Universal Robots PolyScope program: venosa draft3.urp

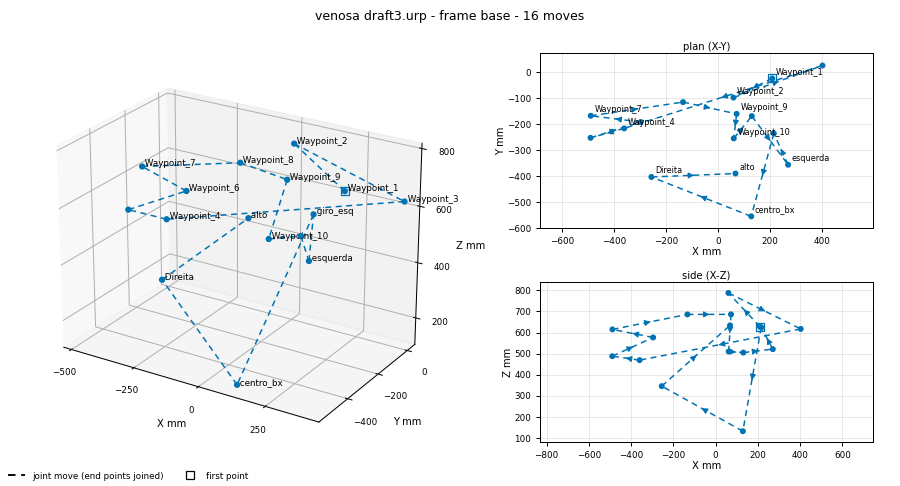
[picture p0: tool path of venosa draft3.urp in frame base, 16 of 16 moves have a stored position in this frame; points joined in program order, loops and branches not executed]
Program venosa draft3 (installation=default directory=/programs/usbdisk createdIn=3.10.1.76190 lastSavedIn=3.10.1.76190 robotSerialNumber=2016331323)
Calibrated DH parameters: a=[0.000045, -0.243749, -0.203764, -0.000005, 0.000123, 0]; d=[0.152024, -1.672567, 11.732654, -9.94768, 0.085297, 0.082386]; alpha=[1.569842, 0.003628, 0.006344, 1.57195, -1.572092, 0]; deltaTheta=[0.000055, -0.024957, 0.328359, -0.303533, 0.000075, 0.000016]
Robot Program (runOnlyOnce=false)
  Folder Danca
    Loop While (checkContinuously=true) expression=Video≟ False
      MoveJ speed 40 deg/s, acceleration 80 deg/s^2 (useActiveTCP=true)
        Waypoint Waypoint_1: TCP in base x=209.295 y=-23.76 z=627.936 mm, rx=0.0536 ry=-0.3833 rz=0.5202 rad; joints [25.586, -182.4, 88.65, -154.413, -90.664, 229.976] deg; flange x=323.162 y=32.336 z=463.353 mm, rx=0.1944 ry=-0.3308 rz=-0.2551 rad
        Waypoint Waypoint_2: TCP in base x=60.121 y=-97.481 z=787.258 mm, rx=-0.0001 ry=-0.0541 rz=0.5161 rad; joints [24.917, -126.62, 79.543, -219.971, -90.664, 229.975] deg; flange x=119.579 y=-66.85 z=590.467 mm, rx=0.0204 ry=-0.0496 rz=-0.2687 rad
        Waypoint Waypoint_3: TCP in base x=402.472 y=25.799 z=616.927 mm, rx=-0.0697 ry=-0.0925 rz=0.3622 rad; joints [17.187, -135.525, -41.809, -87.947, -93.999, 228.948] deg; flange x=475.681 y=35.703 z=422.653 mm, rx=-0.0291 ry=-0.1124 rz=-0.4219 rad
        Waypoint Waypoint_4: TCP in base x=-360.047 y=-215.964 z=469.186 mm, rx=0.079 ry=-1.1865 rz=0.2861 rad; joints [17.753, 2.71, -116.283, -88.686, -94.003, 228.949] deg; flange x=-160.208 y=-163.762 z=445.963 mm, rx=0.5289 ry=-1.0702 rz=-0.4044 rad
        Waypoint Waypoint_5: TCP in base x=-489.412 y=-252.244 z=487.887 mm, rx=0.073 ry=-1.1553 rz=0.2787 rad; joints [17.137, 2.694, -78.551, -128.171, -93.991, 228.95] deg; flange x=-289.897 y=-202.079 z=458.266 mm, rx=0.5117 ry=-1.0443 rz=-0.4168 rad
        Waypoint Waypoint_6: TCP in base x=-296.12 y=-191.355 z=576.602 mm, rx=0.0579 ry=-1.0832 rz=0.2879 rad; joints [17.15, -21.94, -102.997, -83.298, -93.994, 228.949] deg; flange x=-99.068 y=-142.519 z=532.045 mm, rx=0.4698 ry=-0.983 rz=-0.4188 rad
        Waypoint Waypoint_7: TCP in base x=-488.569 y=-167.36 z=614.619 mm, rx=-0.0136 ry=-1.2623 rz=0.131 rad; joints [8.254, -35.552, -41.209, -121.068, -93.991, 228.947] deg; flange x=-281.667 y=-148.953 z=607.37 mm, rx=0.4769 ry=-1.188 rz=-0.546 rad
        Waypoint Waypoint_8: TCP in base x=-133.685 y=-114.831 z=685.693 mm, rx=-0.0287 ry=-1.1088 rz=0.1472 rad; joints [8.292, -74.647, -62.125, -69.9, -93.994, 228.943] deg; flange x=69.715 y=-97.233 z=646.726 mm, rx=0.4031 ry=-1.0497 rz=-0.555 rad
        Waypoint Waypoint_9: TCP in base x=72.457 y=-160.105 z=685.924 mm, rx=0.6935 ry=-0.9793 rz=1.2875 rad; joints [81.88, -74.701, -62.13, -69.92, -93.995, 228.945] deg; flange x=113.042 y=39.927 z=646.676 mm, rx=0.9523 ry=-0.5998 rz=0.5937 rad
        Waypoint Waypoint_10: TCP in base x=61.419 y=-254.47 z=510.056 mm, rx=0.7318 ry=-1.0148 rz=1.2772 rad; joints [81.943, -35.981, -123.832, -44.204, -93.737, 228.945] deg; flange x=100.508 y=-52.476 z=480.549 mm, rx=0.9985 ry=-0.617 rz=0.5916 rad
    Script: stopj(2)
  Folder Rotina Video
    MoveJ speed 75 deg/s, acceleration 80 deg/s^2 (useActiveTCP=true)
      Waypoint inicio_do_filme: TCP in base x=130.91 y=-168.681 z=504.906 mm, rx=1.1521 ry=-1.1466 rz=1.3999 rad; joints [96.272, -151.875, 95.837, -130.575, -90.635, 229.975] deg; flange x=106.895 y=35.088 z=538.092 mm, rx=1.3923 ry=-0.5731 rz=0.7847 rad
      Set DigitalOutput pin=digital_out[1]; digitalValue=1
      SuppressedNode
        Wait Undefined
      Waypoint esquerda: motionParameters(blendRadius=0.05); TCP in base x=270.407 y=-355.692 z=521.272 mm, rx=1.367 ry=-1.0817 rz=1.4077 rad; joints [126.957, -91.39, 65.872, -155.635, -112.651, 225.549] deg; flange x=220.832 y=-160.865 z=574.041 mm, rx=1.55 ry=-0.4405 rz=0.8191 rad
      Waypoint giro_esq: motionParameters(blendRadius=0.05); TCP in base x=215.327 y=-235.3 z=624.251 mm, rx=0.4941 ry=-2.0809 rz=2.158 rad; joints [130.532, -108.88, 55.985, -127.896, -120.939, 297.181] deg; flange x=130.084 y=-46.309 z=638.942 mm, rx=1.0825 ry=-1.4985 rz=1.6715 rad
      Waypoint centro_bx: motionParameters(blendRadius=0.05); TCP in base x=128.595 y=-554.173 z=132.956 mm, rx=0.896 ry=-0.9222 rz=1.5068 rad; joints [88.971, -9.764, 81.203, -275.813, -86.317, 231.862] deg; flange x=111.353 y=-349.34 z=102.199 mm, rx=1.0892 ry=-0.47 rz=0.8261 rad
      Waypoint Direita: motionParameters(blendRadius=0.05); TCP in base x=-255.278 y=-402.824 z=346.182 mm, rx=1.4515 ry=-1.0223 rz=1.5224 rad; joints [4.338, -51.487, 59.787, -182.519, 17.482, 221.464] deg; flange x=-331.706 y=-216.62 z=398.017 mm, rx=1.5869 ry=-0.3567 rz=0.9407 rad
      Waypoint alto: motionParameters(blendRadius=0.05); TCP in base x=67.796 y=-389.459 z=633.759 mm, rx=1.3589 ry=-1.0614 rz=1.299 rad; joints [4.382, -101.171, 18.512, -92.684, 6.521, 216.745] deg; flange x=35.286 y=-191.626 z=688.58 mm, rx=1.5485 ry=-0.4295 rz=0.7067 rad
    Set DigitalOutput pin=vid_fim; digitalValue=1
    Set DigitalOutput pin=digital_out[1]; digitalValue=0
